PROGRAM p_call_fast_task
VAR
	EfficientIO: INT;
END_VAR

(* Es wird standartmäßig M-Bus verwendet, bei IMMODO wurden Mod-Bus zähler verbaut *)
//Communication_KL6781();
(*MAIN_Zaehlerbaustein()*);

(*FB's von Lynus die den FastTask bennötigen*)
EfficientIO_Read_Wirte();

END_PROGRAM

(* stored: Version 1.1.0.1, ProductVersion 3.1.4024.3
   POU p_call_fast_task: Id {a829a65b-3c12-425e-b440-fb072973ae10}, SpecialFunc None *)
